// TIA Portal V20 export
DATA_BLOCK "CallEquipment_DB"   // DB42
{ DB_Accessible_From_OPC_UA := 'FALSE' }
// stored: AssignedProDiagFB Unit1.Em5.ProDiag, DBAccessibleFromOPCUA false, DBAccessibleFromWebserver false, InstanceOfName Unit1.Em5.CallEquipment, InstanceOfType FB, Namespace Unit1.Em5
"Unit1.Em5.CallEquipment"
   // VAR_INPUT
   //    ZoneOperationEnable { ExternalWritable := 'False'} : "LWONIK_typeSafetyZoneManualOperation";
   // END_VAR
   // VAR_IN_OUT
   //    unitStatus : "LAF_typeUnitStatus";
   //    emFeedback : "LUC_typeEmFeedback";
   //    unitAlarmDB : "LAF_typeAlarms";
   // END_VAR
   // VAR
   //    InstSequenceTransferPnPLeft { ExternalWritable := 'False'} : "Unit1.Em5.Sequence_1_TransferPnPLeft";
   //    InstSequenceTransferPnPRight { ExternalWritable := 'False'} : "Unit1.Em5.Sequence_2_TransferPnPRight";
   //    InstSequenceGaugeRnR { ExternalWritable := 'False'} : "Unit1.Em5.Sequence_10_GaugeRnR";
   //    instTransferPnPLeftHomeJob1 { ExternalWritable := 'False'} : "LAF_SelectJob";
   //    instTransferPnPLeftSideTapeLoadJob2 { ExternalWritable := 'False'} : "LAF_SelectJob";
   //    instTransferPnPLeftHotPressLeftUnloadJob3 { ExternalWritable := 'False'} : "LAF_SelectJob";
   //    instTransferPnPLeftHotPressLeftLoadJob4 { ExternalWritable := 'False'} : "LAF_SelectJob";
   //    instTransferPnPLeftSideTapeLoadJob5 { ExternalWritable := 'False'} : "LAF_SelectJob";
   //    instTransferPnPLeftHotPressRightUnloadJob6 { ExternalWritable := 'False'} : "LAF_SelectJob";
   //    instTransferPnPLeftHotPressRightLoadJob7 { ExternalWritable := 'False'} : "LAF_SelectJob";
   //    instTransferPnPLeftHipotThicknessUnloadJob9 { ExternalWritable := 'False'} : "LAF_SelectJob";
   //    instTransferPnPRightHomeJob1 { ExternalWritable := 'False'} : "LAF_SelectJob";
   //    instTransferPnPRightHipotThicknessLoadJob2 { ExternalWritable := 'False'} : "LAF_SelectJob";
   //    instTransferPnPRightVisionUnloadJob3 { ExternalWritable := 'False'} : "LAF_SelectJob";
   //    instTransferPnPRightVisionLoadJob4 { ExternalWritable := 'False'} : "LAF_SelectJob";
   //    instTransferPnPRightLaserMarkUnloadJob5 { ExternalWritable := 'False'} : "LAF_SelectJob";
   //    instTransferPnPRightLaserMarkLoadJob6 { ExternalWritable := 'False'} : "LAF_SelectJob";
   //    instTransferPnPRightWeightCheckUnloadJob9 { ExternalWritable := 'False'} : "LAF_SelectJob";
   //    instGRnR_SideTapeLoadJob2_Left { ExternalWritable := 'False'} : "LAF_SelectJob";
   //    instGRnR_HipotThicknessUnloadJob3_Left { ExternalWritable := 'False'} : "LAF_SelectJob";
   //    instGRnR_HipotThicknessLoadJob4_Left { ExternalWritable := 'False'} : "LAF_SelectJob";
   //    instGRnR_HipotThicknessLoadJob5_Right { ExternalWritable := 'False'} : "LAF_SelectJob";
   //    instGRnR_VisionUnloadJob6_Right { ExternalWritable := 'False'} : "LAF_SelectJob";
   //    instGRnR_VisionLoadJob7_Right { ExternalWritable := 'False'} : "LAF_SelectJob";
   //    instGRnR_WeightCheckUnloadJob8_Right { ExternalWritable := 'False'} : "LAF_SelectJob";
   //    instGRnR_WeightCheckLoadJob9_Right { ExternalWritable := 'False'} : "LAF_SelectJob";
   //    instCmTransferPnPLeftSafetyPin { ExternalWritable := 'False'} : "LBC_DigitalSignalCn";
   //    instCmTransferPnPLeftJRDetect { ExternalWritable := 'False'} : "LBC_DigitalSignalCn";
   //    instCmTransferPnPRightSafetyPin { ExternalWritable := 'False'} : "LBC_DigitalSignalCn";
   //    instCmTransferPnPRightJRDetect { ExternalWritable := 'False'} : "LBC_DigitalSignalCn";
   //    instCmTransferPnPLeftAxisX { ExternalWritable := 'False'} : "LBC_Axis64Pos_TecPlcCn";
   //    instCmTransferPnPLeftAxisY { ExternalWritable := 'False'} : "LBC_Axis64Pos_TecPlcCn";
   //    instCmTransferPnPLeftAxisZ { ExternalWritable := 'False'} : "LBC_Axis64Pos_TecPlcCn";
   //    instCmTransferPnPRightAxisX { ExternalWritable := 'False'} : "LBC_Axis64Pos_TecPlcCn";
   //    instCmTransferPnPRightAxisY { ExternalWritable := 'False'} : "LBC_Axis64Pos_TecPlcCn";
   //    instCmTransferPnPRightAxisZ { ExternalWritable := 'False'} : "LBC_Axis64Pos_TecPlcCn";
   //    instCmTransferPnPLeftClampOpenClose { ExternalWritable := 'False'} : "LBC_TwoWayActuatorCn";
   //    instCmTransferPnPRightClampOpenClose { ExternalWritable := 'False'} : "LBC_TwoWayActuatorCn";
   //    instInterlockTransferPnPLeftAxisX { ExternalWritable := 'False'} : "LER_Axis64Pos_InterlockSummary";
   //    instInterlockTransferPnPLeftAxisY { ExternalWritable := 'False'} : "LER_Axis64Pos_InterlockSummary";
   //    instInterlockTransferPnPLeftAxisZ { ExternalWritable := 'False'} : "LER_Axis64Pos_InterlockSummary";
   //    instInterlockTransferPnPRightAxisX { ExternalWritable := 'False'} : "LER_Axis64Pos_InterlockSummary";
   //    instInterlockTransferPnPRightAxisY { ExternalWritable := 'False'} : "LER_Axis64Pos_InterlockSummary";
   //    instInterlockTransferPnPRightAxisZ { ExternalWritable := 'False'} : "LER_Axis64Pos_InterlockSummary";
   //    instLDrv701ControlTransferPnPLeftAxisZ { ExternalWritable := 'False'} : "LDrvSafe_SinaTlg701Control";
   //    instLDrv701StatusTransferPnPLeftAxisZ { ExternalWritable := 'False'} : "LDrvSafe_SinaTlg701Status";
   //    instLDrv701ControlTransferPnPRightAxisZ { ExternalWritable := 'False'} : "LDrvSafe_SinaTlg701Control";
   //    instLDrv701StatusTransferPnPRightAxisZ { ExternalWritable := 'False'} : "LDrvSafe_SinaTlg701Status";
   //    instManageAlarms { ExternalWritable := 'False'} : "LAF_ManageAlarms";
   //    instEventsPFE { ExternalWritable := 'False'} : "Unit1.Em5.EventsPFE";
   //    statUnitStatus { ExternalWritable := 'False'} : "LAF_typeUnitStatus";
   //    statSlmStatus { ExternalWritable := 'False'} : Struct
   //       running : Bool;
   //       powerOff : Bool;
   //    END_STRUCT;
   //    statAllBrakeTest { ExternalWritable := 'False'} : "LER_typeBrakeTestUnitCommands";
   //    statFlipFlop { ExternalWritable := 'False'} : Array[0..99] of Bool;
   //    statPartData { ExternalWritable := 'False'} : "LER_typePartData";
   //    statDataDelete { ExternalWritable := 'False'} : "LER_typePartData";
   //    statRoutingOk { ExternalWritable := 'False'} : Array[0..99] of Bool;
   //    statRoutingNok { ExternalWritable := 'False'} : Array[0..99] of Bool;
   //    statTonTime { ExternalWritable := 'False'} : Array[0..999] of TON_TIME;
   //    statTofTime { ExternalWritable := 'False'} : Array[0..99] of TOF_TIME;
   //    statPulse { ExternalWritable := 'False'} : Array[0..999] of Bool;
   //    statTrPnP_GaugeRnR : Struct
   //       currentCount : Int;
   //       processCount : Int := 10;
   //       Ongoing : Bool;
   //       Complete : Bool;
   //    END_STRUCT;
   //    statEnableManualCmds { ExternalWritable := 'False'} : Bool;
   //    "*** Interlock Axis ***" : Bool;
   //    TransferPnPLeftAxisX_Home { S7_SetPoint := 'True'} : "LER_Axis_Homing";
   //    TransferPnPLeftAxisY_Home { S7_SetPoint := 'True'} : "LER_Axis_Homing";
   //    TransferPnPLeftAxisZ_Home { S7_SetPoint := 'True'} : "LER_Axis_Homing";
   //    TransferPnPRightAxisX_Home { S7_SetPoint := 'True'} : "LER_Axis_Homing";
   //    TransferPnPRightAxisY_Home { S7_SetPoint := 'True'} : "LER_Axis_Homing";
   //    TransferPnPRightAxisZ_Home { S7_SetPoint := 'True'} : "LER_Axis_Homing";
   //    TransferPnPLeftAxisX_IntHome : Array[0..9] of Bool;
   //    TransferPnPLeftAxisY_IntHome : Array[0..9] of Bool;
   //    TransferPnPLeftAxisZ_IntHome : Array[0..9] of Bool;
   //    TransferPnPRightAxisX_IntHome : Array[0..9] of Bool;
   //    TransferPnPRightAxisY_IntHome : Array[0..9] of Bool;
   //    TransferPnPRightAxisZ_IntHome : Array[0..9] of Bool;
   //    TransferPnPLeftAxisX_Jog { S7_SetPoint := 'True'} : Array[0..2] of "LER_Axis_Jog";
   //    TransferPnPLeftAxisY_Jog { S7_SetPoint := 'True'} : Array[0..2] of "LER_Axis_Jog";
   //    TransferPnPLeftAxisZ_Jog { S7_SetPoint := 'True'} : Array[0..2] of "LER_Axis_Jog";
   //    TransferPnPRightAxisX_Jog { S7_SetPoint := 'True'} : Array[0..2] of "LER_Axis_Jog";
   //    TransferPnPRightAxisY_Jog { S7_SetPoint := 'True'} : Array[0..2] of "LER_Axis_Jog";
   //    TransferPnPRightAxisZ_Jog { S7_SetPoint := 'True'} : Array[0..2] of "LER_Axis_Jog";
   //    TransferPnPLeftAxisX_interlock { S7_SetPoint := 'True'} : Array[0..10] of "LER_Axis_Absolute";
   //    TransferPnPLeftAxisY_interlock { S7_SetPoint := 'True'} : Array[0..10] of "LER_Axis_Absolute";
   //    TransferPnPLeftAxisZ_interlock { S7_SetPoint := 'True'} : Array[0..10] of "LER_Axis_Absolute";
   //    TransferPnPRightAxisX_interlock { S7_SetPoint := 'True'} : Array[0..10] of "LER_Axis_Absolute";
   //    TransferPnPRightAxisY_interlock { S7_SetPoint := 'True'} : Array[0..10] of "LER_Axis_Absolute";
   //    TransferPnPRightAxisZ_interlock { S7_SetPoint := 'True'} : Array[0..10] of "LER_Axis_Absolute";
   //    TransferPnPLeftAxisX_IntPos : Array[0..9] of Struct
   //       "Int" : Array[1..10] of Bool;
   //    END_STRUCT;
   //    TransferPnPLeftAxisY_IntPos : Array[0..9] of Struct
   //       "Int" : Array[1..10] of Bool;
   //    END_STRUCT;
   //    TransferPnPLeftAxisZ_IntPos : Array[0..9] of Struct
   //       "Int" : Array[1..10] of Bool;
   //    END_STRUCT;
   //    TransferPnPRightAxisX_IntPos : Array[0..9] of Struct
   //       "Int" : Array[1..10] of Bool;
   //    END_STRUCT;
   //    TransferPnPRightAxisY_IntPos : Array[0..9] of Struct
   //       "Int" : Array[1..10] of Bool;
   //    END_STRUCT;
   //    TransferPnPRightAxisZ_IntPos : Array[0..9] of Struct
   //       "Int" : Array[1..10] of Bool;
   //    END_STRUCT;
   //    "*** Interlock TwoWay ***" { S7_SetPoint := 'True'} : "LER_Axis_Homing";
   //    instCmTransferPnPLeftClampOpenCloseInterlock { S7_SetPoint := 'True'} : Array[0..2] of "LER_Actuator";
   //    instCmTransferPnPRightClampOpenCloseInterlock { S7_SetPoint := 'True'} : Array[0..2] of "LER_Actuator";
   //    TransferPnPLeftClampOpenClose_Inpos : Array[0..2] of Struct
   //       "Int" : Array[1..10] of Bool;
   //    END_STRUCT;
   //    TransferPnPRightClampOpenClose_Inpos : Array[0..2] of Struct
   //       "Int" : Array[1..10] of Bool;
   //    END_STRUCT;
   //    citi_Ptrig : Array[0..20] of Bool;
   //    citiTon : Array[0..20] of TON_TIME;
   //    citi : Time;
   //    citiTest : Array[0..20] of Bool;
   // END_VAR
BEGIN
END_DATA_BLOCK
